(* IEC 61131-3 sources: crb-codesys/generation/scripts/repoeval/重型运输系统/modbus/PRG, 8 files *)

(* ---- ModbusAct.st ---- *)
PROGRAM ModbusAct
VAR
	bInit					: BOOL:=TRUE;
	iCountAct				: UINT:=10;
	connectStatus			: UINT;
	iErrCode				: BYTE;
	idx						: INT;
	logicIdx				: INT;
	gi						: INT;
	si						: INT;
	iSec					: INT;		//section iterator
	devNum					: WORD;
	fbModbusServer			: ModbusServer;
	inputBuff				: ARRAY[0..1000]OF WORD;
	holdingBuff				: ARRAY[0..1000]OF WORD;

	fbModbusClient			: ModbusTcp_Client;
	fbReadHoldRegister  	: ReadHoldRegister;		//读保持寄存器
	fbWriteMutiRegister		: WriteMutiRegister;
	l2p						: mdbsLogicToPhy;
	p2l						: mdbsPhyToLogic;
	n2i						: mdbsNumToIdx;
	rvs						: DataReverse;
END_VAR

//初始化
IF bInit THEN
	initialize();
	bInit := FALSE;
END_IF

IF connectStatus <> 1 THEN
	fbModbusClient(sIPAddress:='192.168.2.21',uiPort:=520);//连接IPC
	//fbModbusClient(sIPAddress:='192.168.5.55',uiPort:=502);//连接工控机
END_IF

IF fbModbusClient.bSuccess THEN
	connectStatus := 1;
	CASE iCountAct OF
		10:
			handleCmd();		//接收华中指令
			localCmdHandler();	//处理本机挡板指令 + 启动液压站
		20:
			handleStat1();		//发送状态至华中
		21:
			handleStat2();
		22:
			handleStat3();
	END_CASE
END_IF

//做服务器接收天地轨客户端发送的数据
fbModbusServer(	wPort := 512,
	pInputData := ADR(inputBuff[0]), pOutputData := ADR(holdingBuff[0]),
	uiInputDataSize := 1000, uiOutputDataSize := 1000,
	xEnable := TRUE, xReset := FALSE, tTimeout := 1000,
	xBusy => , xError => , byClientConnections => );

//将缓冲区Buff数据转至本地
localStatHandler();
//updateStat();

(* ---- ModbusAct_handleCmd.st ---- *)
fbReadHoldRegister(
	xExecute	:= TRUE,
	slaveId		:= 1,
	wStartAdr	:= gModbus.srv.request.startAddr,
	wLen		:= gModbus.srv.request.length,
	pTcpStream	:= fbModbusClient.pfbTcpStream,
	modbusHoldRegData:= gModbus.modbusBuffer);

IF fbReadHoldRegister.bSucced THEN
	fbReadHoldRegister(xExecute := FALSE,
						modbusHoldRegData:=g_modbusHoldRegData);

	//使用holdingBuff接收供给链控制指令，在下一轮循环中作为服务器保持该数据
	FOR idx := 10 TO 57 DO			//startAddr to startAddr+length-1
		holdingBuff[idx] := gModbus.modbusBuffer[idx];
	END_FOR

	iCountAct := 20;
END_IF

IF fbReadHoldRegister.berror THEN
	fbReadHoldRegister(xExecute :=FALSE,
						modbusHoldRegData:= gModbus.modbusBuffer);
	fbModbusClient.M_Reset();
	connectStatus := 0;
	iCountAct := 10;
	iErrCode := fbReadHoldRegister.errCode;
END_IF

(* ---- ModbusAct_handleStat1.st ---- *)
fbWriteMutiRegister(
	xExecute	:= TRUE,
	slaveId		:= 1,
	startAddr	:= 110, //gModbus.srv.response.startAddr 110-319
	wRegNum		:= 70,
	value		:= ADR(gModbus.srv.response.data[110]),
	pTcpStream	:= fbModbusClient.pfbTcpStream);

IF fbWriteMutiRegister.bSucced THEN
	fbWriteMutiRegister(xExecute := FALSE);
	iCountAct:= 21;
END_IF

IF fbWriteMutiRegister.berror THEN
	fbWriteMutiRegister(xExecute := FALSE);
	fbModbusClient.M_Reset();
	iCountAct := 10;
	connectStatus := 0;
	iErrCode := fbWriteMutiRegister.errCode;
END_IF

(* ---- ModbusAct_handleStat2.st ---- *)
fbWriteMutiRegister(
	xExecute	:= TRUE,
	slaveId		:= 1,
	startAddr	:= 180, //gModbus.srv.response.startAddr 110-319
	wRegNum		:= 70,
	value		:= ADR(gModbus.srv.response.data[180]),
	pTcpStream	:= fbModbusClient.pfbTcpStream);

IF fbWriteMutiRegister.bSucced THEN
	fbWriteMutiRegister(xExecute := FALSE);
	iCountAct:= 22;
END_IF

IF fbWriteMutiRegister.berror THEN
	fbWriteMutiRegister(xExecute := FALSE);
	fbModbusClient.M_Reset();
	iCountAct := 10;
	connectStatus := 0;
	iErrCode := fbWriteMutiRegister.errCode;
END_IF

(* ---- ModbusAct_handleStat3.st ---- *)
fbWriteMutiRegister(
	xExecute	:= TRUE,
	slaveId		:= 1,
	startAddr	:= 250, //gModbus.srv.response.startAddr 110-319
	wRegNum		:= 70,
	value		:= ADR(gModbus.srv.response.data[250]),
	pTcpStream	:= fbModbusClient.pfbTcpStream);

IF fbWriteMutiRegister.bSucced THEN
	fbWriteMutiRegister(xExecute := FALSE);
	iCountAct:= 10;
END_IF

IF fbWriteMutiRegister.berror THEN
	fbWriteMutiRegister(xExecute := FALSE);
	fbModbusClient.M_Reset();
	iCountAct := 10;
	connectStatus := 0;
	iErrCode := fbWriteMutiRegister.errCode;
END_IF

(* ---- ModbusAct_localCmdHandler.st ---- *)
METHOD localCmdHandler
VAR_INPUT
END_VAR
VAR
	iBit				:INT;
	exLevel				:INT;
	exIdx				:INT;
	exDirect			:TargetDirect;
	exeDirect			:TargetDirect;

END_VAR
VAR CONSTANT
	no		:ARRAY [1..8] OF INT :=[11, 14, 17, 20, 49, 50, 51, 52];
END_VAR

FOR iSec := 1 TO 8 DO
	gModbus.srv.request.data[no[iSec]] := gModbus.modbusBuffer[no[iSec]];
END_FOR

FOR iSec := 1 TO 4 DO
	gModbus.srv.request.arrNew[iSec,1	] := gModbus.srv.request.data[no[iSec]].1	;
	gModbus.srv.request.arrNew[iSec,2	] := gModbus.srv.request.data[no[iSec]].2	;
	gModbus.srv.request.arrNew[iSec,3	] := gModbus.srv.request.data[no[iSec]].3	;
	gModbus.srv.request.arrNew[iSec,4	] := gModbus.srv.request.data[no[iSec]].4	;
	gModbus.srv.request.arrNew[iSec,5	] := gModbus.srv.request.data[no[iSec]].5	;
	gModbus.srv.request.arrNew[iSec,6	] := gModbus.srv.request.data[no[iSec]].6	;
	gModbus.srv.request.arrNew[iSec,7	] := gModbus.srv.request.data[no[iSec]].7	;
	gModbus.srv.request.arrNew[iSec,8	] := gModbus.srv.request.data[no[iSec]].8	;
	gModbus.srv.request.arrNew[iSec,9	] := gModbus.srv.request.data[no[iSec]].9	;
	gModbus.srv.request.arrNew[iSec,10	] := gModbus.srv.request.data[no[iSec]].10	;
	gModbus.srv.request.arrNew[iSec,11	] := gModbus.srv.request.data[no[iSec]].11	;
END_FOR
FOR iSec := 1 TO 4 DO
	FOR iBit := 1 TO 11 DO
		IF gModbus.srv.request.arrNew[iSec, iBit] <> gModbus.srv.request.arrLast[iSec, iBit] THEN
			IF gModbus.srv.request.arrNew[iSec, iBit] THEN	//仅执行上升沿
				//specifically output[grd/sky(exLevel), no(exIdx), TargetDirect(exDirect)]
				l2p(section := iSec, lgcIdx := iBit,
					level => exLevel, phyIdx => exIdx, direct => exDirect);
				exeDirect := rvs.cmdReverse(input := exDirect);		//华中要求伸缩指令及状态翻转

				//过滤	机械结构未完成的grd[4] and sky[4]
				IF exIdx = 4 THEN	exeDirect := TargetDirect.stop;	END_IF

				setButtonByDirect(level := exLevel, idx := exIdx, direct := exeDirect);
			END_IF
			gModbus.srv.request.arrLast[iSec, iBit] := gModbus.srv.request.arrNew[iSec, iBit];
		END_IF
	END_FOR

END_FOR

devNum := gModbus.modbusBuffer[49];

//新增一键启动液压站

IF gUI.mode.hydPowerOn THEN
	holdingBuff[48] := holdingBuff[48] OR 1;
END_IF
IF gUI.mode.hydPowerOff THEN
	holdingBuff[48] := holdingBuff[48] OR 2;
END_IF

(* ---- ModbusAct_localStatHandler.st ---- *)
METHOD localStatHandler : TargetDirect
VAR_INPUT
END_VAR

//先把天地轨控制器数据同步至本地
FOR idx := 110 TO 319 DO
	gModbus.srv.response.data[idx] := holdingBuff[idx];
END_FOR

//根据实际状态将挡板数据同步至本地
FOR gi := 1 TO 10 DO
	(*******************************
	伸缩反向判定，伸出到位返回缩回到位
	**********************************)

	//地轨伸出到位检查
	p2l(section := 1, phyIdx := gi, lgcIdx => logicIdx);//logicIdx范围[223,232]
	IF gDev.grd[gi].state = DevStatus.retracted THEN
		gModbus.srv.response.data[logicIdx] := 1;
	ELSE
		gModbus.srv.response.data[logicIdx] := 0;
	END_IF
	//地轨缩回到位检查
	p2l(section := 2, phyIdx := gi, lgcIdx => logicIdx);//logicIdx范围[271,280]
	IF gDev.grd[gi].state = DevStatus.extended THEN
		gModbus.srv.response.data[logicIdx] := 1;
	ELSE
		gModbus.srv.response.data[logicIdx] := 0;
	END_IF
END_FOR

FOR si := 0 TO 10 DO
	//天轨伸出到位检查
	p2l(section := 3, phyIdx := si, lgcIdx => logicIdx);//logicIdx范围[127,137]

	IF gDev.sky[si].state = DevStatus.retracted THEN
		gModbus.srv.response.data[logicIdx] := 1;
	ELSE
		gModbus.srv.response.data[logicIdx] := 0;
	END_IF
	//天轨缩回到位检查
	p2l(section := 4, phyIdx := si, lgcIdx => logicIdx);//logicIdx范围[175,185]
	IF gDev.sky[si].state = DevStatus.extended THEN
		gModbus.srv.response.data[logicIdx] := 1;
	ELSE
		gModbus.srv.response.data[logicIdx] := 0;
	END_IF
END_FOR
//至此110-309寄存器状态更新完毕，向华中发送时只需在寄存器写入response.data[]数组

IF devNum > 40000 THEN
	n2i(devNo := devNum, level => , idx =>);
	CASE n2i.level OF
		1:
			gModbus.srv.response.data[312] := REAL_TO_WORD(10 * gDev.grd[n2i.idx].sensor.position);
			gModbus.srv.response.data[313] := REAL_TO_WORD(10 * gDev.grd[n2i.idx].sensor.extendVal);
			gModbus.srv.response.data[314] := REAL_TO_WORD(10 * gDev.grd[n2i.idx].sensor.retractVal);
		2:
			gModbus.srv.response.data[312] := REAL_TO_WORD(10 * gDev.sky[n2i.idx].sensor.position);
			gModbus.srv.response.data[313] := REAL_TO_WORD(10 * gDev.sky[n2i.idx].sensor.extendVal);
			gModbus.srv.response.data[314] := REAL_TO_WORD(10 * gDev.sky[n2i.idx].sensor.retractVal);
	END_CASE
END_IF

(* ---- ModbusAct_updateStat.st ---- *)
//先把天地轨控制器数据同步至本地
FOR idx := 110 TO 319 DO
	gModbus.srv.response.data[idx] := holdingBuff[idx];
END_FOR

//根据实际状态将挡板数据同步至本地
FOR gi := 1 TO 10 DO

	//地轨伸出到位检查
	p2l(section := 1, phyIdx := gi, lgcIdx => logicIdx);//logicIdx范围[223,232]
	IF gDev.grd[gi].state = DevStatus.extended THEN
		gModbus.srv.response.data[logicIdx] := 1;
	ELSE
		gModbus.srv.response.data[logicIdx] := 0;
	END_IF
	//地轨缩回到位检查
	p2l(section := 2, phyIdx := gi, lgcIdx => logicIdx);//logicIdx范围[271,280]
	IF gDev.grd[gi].state = DevStatus.retracted THEN
		gModbus.srv.response.data[logicIdx] := 1;
	ELSE
		gModbus.srv.response.data[logicIdx] := 0;
	END_IF
END_FOR

FOR si := 0 TO 10 DO
	//天轨伸出到位检查
	p2l(section := 3, phyIdx := si, lgcIdx => logicIdx);//logicIdx范围[127,137]
	IF gDev.sky[si].state = DevStatus.extended THEN
		gModbus.srv.response.data[logicIdx] := 1;
	ELSE
		gModbus.srv.response.data[logicIdx] := 0;
	END_IF
	//天轨缩回到位检查
	p2l(section := 4, phyIdx := si, lgcIdx => logicIdx);//logicIdx范围[175,185]
	IF gDev.sky[si].state = DevStatus.retracted THEN
		gModbus.srv.response.data[logicIdx] := 1;
	ELSE
		gModbus.srv.response.data[logicIdx] := 0;
	END_IF
END_FOR
//至此110-309寄存器状态更新完毕，向华中发送时只需在寄存器写入response.data[]数组

IF devNum > 40000 THEN
	n2i(devNo := devNum, level => , idx =>);
	CASE n2i.level OF
		1:
			gModbus.srv.response.data[312] := REAL_TO_WORD(10 * gDev.grd[n2i.idx].sensor.position);
			gModbus.srv.response.data[313] := REAL_TO_WORD(10 * gDev.grd[n2i.idx].sensor.extendVal);
			gModbus.srv.response.data[314] := REAL_TO_WORD(10 * gDev.grd[n2i.idx].sensor.retractVal);
		2:
			gModbus.srv.response.data[312] := REAL_TO_WORD(10 * gDev.sky[n2i.idx].sensor.position);
			gModbus.srv.response.data[313] := REAL_TO_WORD(10 * gDev.sky[n2i.idx].sensor.extendVal);
			gModbus.srv.response.data[314] := REAL_TO_WORD(10 * gDev.sky[n2i.idx].sensor.retractVal);
	END_CASE
END_IF
